(* PLC project lightclock, Dassault Systèmes ControlBuild 2024x *)
(* stored: creationDateTime 2023-10-03T11:13:47-01:00 *)

FUNCTION_BLOCK tni_clock.lightclock
  VAR_INPUT
    switchOnLight : BOOL := false;
  END_VAR


END_FUNCTION_BLOCK
